FUNCTION Convert_REAL_TO_UINT : Hresult
VAR_INPUT
	in : REAL;
	out : REFERENCE TO UINT;
END_VAR
VAR
	converted : UINT;
END_VAR
VAR CONSTANT
	INCOMPATIBLE : HRESULT := 16#9811070E;
END_VAR

converted := REAL_TO_UINT(in);

IF (UINT_TO_REAL(converted) <> in) THEN
	Convert_REAL_TO_UINT := INCOMPATIBLE;
	RETURN;
END_IF

out := converted;

END_FUNCTION

(* stored: Version 1.1.0.1, ProductVersion 3.1.4024.12
   POU Convert_REAL_TO_UINT: Id {2adc5302-1043-4313-94a4-d10f14b5ed12}, SpecialFunc None *)
